TYPE ST_EndStops :
STRUCT
	sNoEndStop : STRING := 'End Stop not active';
	sPistonUpperEndStop : STRING := 'Piston has reached upper end stop';
	sPistonLowerEndStop : STRING := 'Piston has reached lower end stop';
END_STRUCT
END_TYPE

(* stored: Version 1.1.0.1, ProductVersion 3.1.4024.10
   DUT ST_EndStops: Id {cf9f0ed6-3148-4ebf-9665-44f4664dc3e1} *)
